TYPE DUT_01_Channel_NW :
STRUCT
    header: DUT_Header_NW;
    channel1: DUT_Channel_NW;
END_STRUCT
END_TYPE

(* stored: Version 1.1.0.1, ProductVersion 3.1.4022.18
   DUT DUT_01_Channel_NW: Id {db4ee9da-1d10-4532-b458-8f8787ea5d90} *)
